FUNCTION_BLOCK FB_Stn512DivertTC
VAR_INPUT
	
	pCmp: POINTER TO CmpConvDivert;

END_VAR

VAR
	
	MainRunning: BOOL;
	SpurRunning: BOOL;
	
	onsPuckReady: R_TRIG;
	ResolvedDBStatusRouteBlue: cResolvedDBStatusRoute;
	ResolvedDBStatusRouteGreen: cResolvedDBStatusRoute;
	ResolvedDBStatusRouteRed: cResolvedDBStatusRoute;
	DBRouteToSpur_Empty: BOOL;
	DBRouteToSpur_Full: BOOL;
	RouteToSpur: BOOL;
	
	HoldFullPuck: BOOL;
	
	tmrSpurNotOKToReceive: TON;
	
	Debug_ForceAllApplicableToSpur: BOOL;
	Debug_StationEmptyPuckReq: BOOL;
	Debug_DivertAllToMain: BOOL;
	Debug_DivertAllToSpur: BOOL;
	Debug_AllowHoldFullPuck: BOOL;
	
END_VAR

// Traffic control for specific dirvert - Stn060
// 
// Currently each divert has independent/unique function block as it is expected that they will
//   eventually need to be tweeked for specific application

// Sum of main/spur running conditions... don't release if not running
MainRunning :=
	pCmp^.MainHeartbeatOK AND
	pCmp^.MainConvRunning;

SpurRunning :=
	pCmp^.SpurHeartbeatOK AND
	pCmp^.SpurConvRunning;

// On rising edege of puck ready interperate the puck/device data to see if it should be diverted to spur
onsPuckReady(CLK:=pCmp^.PuckReady);
IF onsPuckReady.Q THEN 	
	// Call function to turn DB puck/device status/route into single readable resolution
	ResolvedDBStatusRouteGreen :=
		FN_ResolveDBStatusRoutePuck(
			Puck := pCmp^.Puck,
			RouteToWork := cDBDetailRoute.TrayLoadGreen);
	ResolvedDBStatusRouteRed :=
		FN_ResolveDBStatusRoutePuck(
			Puck := pCmp^.Puck,
			RouteToWork := cDBDetailRoute.TrayLoadRed);
	ResolvedDBStatusRouteBlue :=
		FN_ResolveDBStatusRoutePuck(
			Puck := pCmp^.Puck,
			RouteToWork := cDBDetailRoute.TrayLoadBlue);
		
	// Use DB route and other possible line status to determine if puck should go to spur
	// This station never works on an empty puck.
	
	DBRouteToSpur_Empty := 
		Debug_StationEmptyPuckReq AND
		(ResolvedDBStatusRouteRed = cResolvedDBStatusRoute.Empty_NoRoute OR
		ResolvedDBStatusRouteRed = cResolvedDBStatusRoute.Empty_RoutedThisStation OR
		ResolvedDBStatusRouteRed = cResolvedDBStatusRoute.Empty_RoutedOtherStation);
	
	DBRouteToSpur_Full := 
		(ResolvedDBStatusRouteBlue = cResolvedDBStatusRoute.Normal_RoutedThisStation OR
			ResolvedDBStatusRouteRed = cResolvedDBStatusRoute.Normal_RoutedThisStation OR
			ResolvedDBStatusRouteGreen = cResolvedDBStatusRoute.Normal_RoutedThisStation) AND
			pCmp^.Puck.Side = TO_STRING(cPuckSide.Clean);
END_IF

RouteToSpur := 
	DBRouteToSpur_Full OR
	(DBRouteToSpur_Empty AND
	Debug_StationEmptyPuckReq) OR
	(Debug_ForceAllApplicableToSpur AND	
	pCmp^.Puck.Side = TO_STRING(cPuckSide.Clean) AND
	pCmp^.Puck.Device.RowaTrayType = cDBRowaTrayType.Small);

	
// Run timer for spur not ok to receive
// TODO - RCC: Eventualy include upstream buffer full before forcing release
tmrSpurNotOKToReceive(
		IN:= NOT SpurRunning OR NOT pCmp^.senSpurBufferFullOff,
		PT:= T#1000MS);
		
// Release main if that is DB route or if spur not ready in time
//  and a few other misc conditions.

pCmp^.PuckReleaseMain := 
	pCmp^.PuckReady AND
	MainRunning AND
	(NOT RouteToSpur OR
	tmrSpurNotOkToReceive.Q OR
	pCmp^.UnknownPuck OR
	Debug_DivertAllToMain) AND
	NOT Debug_DivertAllToSpur;


IF Debug_AllowHoldFullPuck THEN

//HOLD this puck to spur; do not release to main if full puck and is going to spur
	HoldFullPuck := pCmp^.Puck.Device.SN <> '' AND RouteToSpur;
// get upstream BF from previous merge/divert to disable HoldFullPuck feature, to reduce the long wait times and keep some puck flowing
	IF gStn055_46_Stn511MainMergePrestop.StatusBufferFull THEN
		HoldFullPuck := FALSE;
	END_IF

	pCmp^.PuckReleaseMain := pCmp^.PuckReleaseMain AND NOT HoldFullPuck;
END_IF

// Release to spur if that is route and it is available.
pCmp^.PuckReleaseSpur :=
	pCmp^.PuckReady AND
	MainRunning AND
	SpurRunning AND
	((RouteToSpur AND
	NOT pCmp^.UnknownPuck) OR
	Debug_DivertAllToSpur) AND
	NOT Debug_DivertAllToMain;

END_FUNCTION_BLOCK

(* stored: Version 1.1.0.1, ProductVersion 3.1.4024.6
   POU FB_Stn512DivertTC: Id {becff735-7e8e-40a5-be90-2a6132cadbb3}, SpecialFunc None *)
